KUKA KRL program: G1_LI2.src, G1_LI2.dat

--- G1_LI2.src ---
&ACCESS RVO1
&COMMENT
DEF G1_LI2 ( )

STRUC Note real x, y, interval
Note music[100]

music[0].x = 0
music[0].y = 0
music[0].interval = 0

;FOLD INI
  ;FOLD BASISTECH INI
    GLOBAL INTERRUPT DECL 3 WHEN $STOPMESS==TRUE DO IR_STOPM ( )
    INTERRUPT ON 3
    BAS (#INITMOV,0 )
  ;ENDFOLD (BASISTECH INI)
  ;FOLD USER INI
    ;Make your modifications here

  ;ENDFOLD (USER INI)
;ENDFOLD (INI)
LOOP
;FOLD PTP HOME  Vel= 10 % DEFAULT;%{PE}%MKUKATPBASIS,%CMOVE,%VPTP,%P 1:PTP, 2:HOME, 3:, 5:100, 7:DEFAULT
$BWDSTART = FALSE
PDAT_ACT=PDEFAULT
FDAT_ACT=FHOME
BAS (#PTP_PARAMS,100 )
$H_POS=XHOME
PTP  XHOME
;ENDFOLD

;FOLD PTP P1  Vel=10 % PDAT1 Tool[0] Base[0];%{PE}%R 8.3.22,%MKUKATPBASIS,%CMOVE,%VPTP,%P 1:PTP, 2:P1, 3:, 5:100, 7:PDAT1
$BWDSTART=FALSE
PDAT_ACT=PPDAT1
FDAT_ACT=FP1
BAS(#PTP_PARAMS,100)
PTP XP1
;ENDFOLD
WAIT SEC 1

;FOLD PTP P2  Vel=10 % PDAT2 Tool[0] Base[0];%{PE}%R 8.3.22,%MKUKATPBASIS,%CMOVE,%VPTP,%P 1:PTP, 2:P2, 3:, 5:100, 7:PDAT2
$BWDSTART=FALSE
PDAT_ACT=PPDAT2
FDAT_ACT=FP2
BAS(#PTP_PARAMS,100)
PTP XP2
;ENDFOLD
WAIT SEC 1

;FOLD PTP HOME  Vel=10 % DEFAULT;%{PE}%MKUKATPBASIS,%CMOVE,%VPTP,%P 1:PTP, 2:HOME, 3:, 5:100, 7:DEFAULT
$BWDSTART = FALSE
PDAT_ACT=PDEFAULT
FDAT_ACT=FHOME
BAS (#PTP_PARAMS,100 )
$H_POS=XHOME
PTP  XHOME
;ENDFOLD
WAIT SEC 3

;FOLD PTP P2  Vel=10 % PDAT2 Tool[0] Base[0];%{PE}%R 8.3.22,%MKUKATPBASIS,%CMOVE,%VPTP,%P 1:PTP, 2:P2, 3:, 5:100, 7:PDAT2
$BWDSTART=FALSE
PDAT_ACT=PPDAT2
FDAT_ACT=FP2
BAS(#PTP_PARAMS,100)
PTP XP2
;ENDFOLD
WAIT SEC 1

;FOLD PTP P3  Vel=10 % PDAT3 Tool[0] Base[0];%{PE}%R 8.3.22,%MKUKATPBASIS,%CMOVE,%VPTP,%P 1:PTP, 2:P3, 3:, 5:100, 7:PDAT3
$BWDSTART=FALSE
PDAT_ACT=PPDAT3
FDAT_ACT=FP3
BAS(#PTP_PARAMS,100)
PTP XP3
;ENDFOLD
WAIT SEC 1

ENDLOOP
;FOLD PTP HOME  Vel=10 % DEFAULT;%{PE}%MKUKATPBASIS,%CMOVE,%VPTP,%P 1:PTP, 2:HOME, 3:, 5:100, 7:DEFAULT
$BWDSTART = FALSE
PDAT_ACT=PDEFAULT
FDAT_ACT=FHOME
BAS (#PTP_PARAMS,100 )
$H_POS=XHOME
PTP  XHOME
;ENDFOLD

END

--- G1_LI2.dat ---
&ACCESS RVO1
&COMMENT
DEFDAT G1_LI2 PUBLIC
;FOLD EXTERNAL DECLARATIONS;%{PE}%MKUKATPBASIS,%CEXT,%VCOMMON,%P
;FOLD BASISTECH EXT;%{PE}%MKUKATPBASIS,%CEXT,%VEXT,%P
EXT  BAS (BAS_COMMAND  :IN,REAL  :IN )
DECL INT SUCCESS
;ENDFOLD (BASISTECH EXT)
;FOLD USER EXT;%{E}%MKUKATPUSER,%CEXT,%VEXT,%P
;Make here your modifications

;ENDFOLD (USER EXT)
;ENDFOLD (EXTERNAL DECLERATIONS)
DECL BASIS_SUGG_T LAST_BASIS={POINT1[] "P3",POINT2[] "P3",CP_PARAMS[] "CPDAT0",PTP_PARAMS[] "PDAT3",CONT[] " ",CP_VEL[] "2",PTP_VEL[] "100",SYNC_PARAMS[] " ",SPL_NAME[] " "}
DECL E6POS XP1={X 0,Y 0,Z 0,A 0,B 0,C 0,S 0,T 0,E1 0,E2 0,E3 0,E4 0,E5 0,E6 0}
DECL FDAT FP1={TOOL_NO 0,BASE_NO 0,IPO_FRAME #BASE,POINT2[] " ",TQ_STATE FALSE}
DECL PDAT PPDAT1={VEL 100,ACC 100,APO_DIST 100,APO_MODE #CPTP,GEAR_JERK 50}
DECL E6POS XP2={X 0,Y 0,Z 0,A 0,B 0,C 0,S 0,T 0,E1 0,E2 0,E3 0,E4 0,E5 0,E6 0}
DECL FDAT FP2={TOOL_NO 0,BASE_NO 0,IPO_FRAME #BASE,POINT2[] " ",TQ_STATE FALSE}
DECL PDAT PPDAT2={VEL 100,ACC 100,APO_DIST 100,APO_MODE #CPTP,GEAR_JERK 50}
DECL E6POS XP3={X 0,Y 0,Z 0,A 0,B 0,C 0,S 0,T 0,E1 0,E2 0,E3 0,E4 0,E5 0,E6 0}
DECL FDAT FP3={TOOL_NO 0,BASE_NO 0,IPO_FRAME #BASE,POINT2[] " ",TQ_STATE FALSE}
DECL PDAT PPDAT3={VEL 100,ACC 100,APO_DIST 100,APO_MODE #CPTP,GEAR_JERK 50}
ENDDAT
